// Mitsubishi GX Works2 project: operacoes_basicas   PLC: Q03UDV
// turma1

PROGRAM MAIN
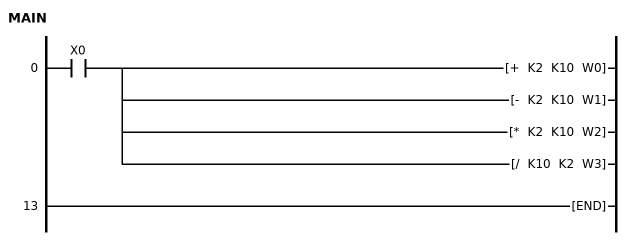
0     LD      X0
      +       K2 K10 W0
      -       K2 K10 W1
      *       K2 K10 W2
      /       K10 K2 W3
13    END
END_PROGRAM
